SUBAPPLICATION Uebung_002a2 (* DigitalInput_I1/_I2 mit AND (alt) auf DigitalOutput_Q1 *)
  (* Standard: 61499-2; Description: Copyright (c) 2023 Meisterschulen am Ostbahnhof This program and the accompanying materials are made available under the terms of the Eclipse Public License 2.0 which is available at https://www.eclipse.org/legal/epl-2.0/ SPDX-License-Identifier: EPL-2.0 *)
  (* Version 1.0, 2023-10-23, Franz Höpfinger, Meisterschulen am Ostbahnhof *)
  PACKAGE Uebungen;
  IMPORT logiBUS::io::DI::logiBUS_DI::Input_I1;
  IMPORT logiBUS::io::DI::logiBUS_DI::Input_I2;
  IMPORT logiBUS::io::DQ::logiBUS_DO::Output_Q1;
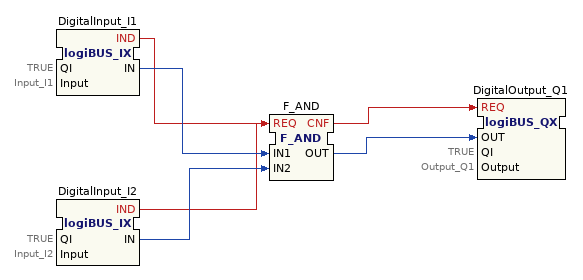
  FBS
    DigitalOutput_Q1 : logiBUS::io::DQ::logiBUS_QX(QI := TRUE, Output := Output_Q1);
    DigitalInput_I1 : logiBUS::io::DI::logiBUS_IX(QI := TRUE, Input := Input_I1);
    DigitalInput_I2 : logiBUS::io::DI::logiBUS_IX(QI := TRUE, Input := Input_I2);
    F_AND : iec61131::bitwiseOperators::F_AND;
  END_FBS
  EVENT_CONNECTIONS
    DigitalInput_I1.IND TO F_AND.REQ;
    DigitalInput_I2.IND TO F_AND.REQ;
    F_AND.CNF TO DigitalOutput_Q1.REQ;
  END_CONNECTIONS
  DATA_CONNECTIONS
    F_AND.OUT TO DigitalOutput_Q1.OUT;
    DigitalInput_I1.IN TO F_AND.IN1;
    DigitalInput_I2.IN TO F_AND.IN2;
  END_CONNECTIONS
END_SUBAPPLICATION
